FUNCTION BufferIntToReal : Real
VAR_INPUT
	raw_input :INT;
END_VAR
VAR
	temp : DWORD;
END_VAR

temp := UDINT_TO_DWORD(raw_input);
BufferUdintToReal := DWORD_TO_REAL(temp);
temp := BE32_TO_HOST(temp);
MEMCPY(ADR(BufferUdintToReal), ADR(temp), SIZEOF(temp));

END_FUNCTION

(* stored: Version 1.1.0.1, ProductVersion 3.1.4024.9
   POU BufferIntToReal: Id {5ba4695c-2ebb-4c7e-85fa-5e012c521cf2}, SpecialFunc None *)
